(* IEC 61131-3 sources: com.logicals.lc3.webinar/logicals_Lib_Webinar/logicals_Webinar_Basic_Lib/logicals_Lib/src_FB_ST/Logic, 1 file *)

(* ---- logicals_Logic_ST.iecst ---- *)
NAMESPACE com.logicals.Basic.Logic

FUNCTION_BLOCK FB_lc_1oo3_ST

  VAR_INPUT
    vix_In1 : BOOL;
    vix_In2 : BOOL;
    vix_In3 : BOOL;
  END_VAR

  VAR_OUTPUT
   vox_Out : BOOL;
  END_VAR

  VAR
   lx_Var_AND1  : BOOL;
   lx_Var_AND2 : BOOL;
   lx_Var_AND3 : BOOL;
  END_VAR

  // Network 1:
  lx_Var_AND1 := AND(IN1 := vix_In1, IN2 := NOT vix_In2, IN3 := NOT vix_In3);
  lx_Var_AND2 := AND(IN1 := NOT vix_In1, IN2 := vix_In2, IN3 := NOT vix_In3);
  lx_Var_AND3 := AND(IN1 := NOT vix_In1, IN2 := NOT vix_In2, IN3 := vix_In3);
  vox_Out := OR(IN1 := lx_Var_AND1, IN2 := lx_Var_AND2, IN3 := lx_Var_AND3);

END_FUNCTION_BLOCK

FUNCTION_BLOCK FB_lc_1oo4_ST
	VAR_INPUT
		vix_In1 : BOOL;
		vix_In2 : BOOL;
		vix_In3 : BOOL;
		vix_In4 : BOOL;
	END_VAR

	VAR_OUTPUT
		vox_Out1 : BOOL;
		vox_Out2 : BOOL;
		vox_Out3 : BOOL;
		vox_Out4 : BOOL;

        vox_Err  : BOOL;
	END_VAR

    vox_Out1 := vix_In1 = TRUE  AND vix_In2 = FALSE AND vix_In3 = FALSE AND vix_In4 = FALSE;
    vox_Out2 := vix_In1 = FALSE AND vix_In2 = TRUE  AND vix_In3 = FALSE AND vix_In4 = FALSE;
    vox_Out3 := vix_In1 = FALSE AND vix_In2 = FALSE AND vix_In3 = TRUE  AND vix_In4 = FALSE;
    vox_Out4 := vix_In1 = FALSE AND vix_In2 = FALSE AND vix_In3 = FALSE AND vix_In4 = TRUE ;

    vox_Err :=  NOT(vox_Out1 = TRUE OR vox_Out2 = TRUE OR vox_Out3 = TRUE OR vox_Out4 = TRUE);

END_FUNCTION_BLOCK

FUNCTION_BLOCK FB_lc_1oo5_ST
	VAR_INPUT
		vix_In1 : BOOL;
		vix_In2 : BOOL;
		vix_In3 : BOOL;
		vix_In4 : BOOL;
		vix_In5 : BOOL;
	END_VAR

	VAR_OUTPUT
		vox_Out1 : BOOL;
		vox_Out2 : BOOL;
		vox_Out3 : BOOL;
		vox_Out4 : BOOL;
		vox_Out5 : BOOL;

        vox_Err  : BOOL;
	END_VAR

    vox_Out1 := vix_In1 = TRUE  AND vix_In2 = FALSE AND vix_In3 = FALSE AND vix_In4 = FALSE AND vix_In5 = FALSE;
    vox_Out2 := vix_In1 = FALSE AND vix_In2 = TRUE  AND vix_In3 = FALSE AND vix_In4 = FALSE AND vix_In5 = FALSE;
    vox_Out3 := vix_In1 = FALSE AND vix_In2 = FALSE AND vix_In3 = TRUE  AND vix_In4 = FALSE AND vix_In5 = FALSE;
    vox_Out4 := vix_In1 = FALSE AND vix_In2 = FALSE AND vix_In3 = FALSE AND vix_In4 = TRUE  AND vix_In5 = FALSE;
    vox_Out5 := vix_In1 = FALSE AND vix_In2 = FALSE AND vix_In3 = FALSE AND vix_In4 = FALSE AND vix_In5 = TRUE;

    vox_Err :=  NOT(vox_Out1 = TRUE OR vox_Out2 = TRUE OR vox_Out3 = TRUE OR vox_Out4 = TRUE OR vox_Out5 = TRUE );

END_FUNCTION_BLOCK

FUNCTION_BLOCK FB_lc_1oo6_ST
	VAR_INPUT
		vix_In1 : BOOL;
		vix_In2 : BOOL;
		vix_In3 : BOOL;
		vix_In4 : BOOL;
		vix_In5 : BOOL;
		vix_In6 : BOOL;
	END_VAR

	VAR_OUTPUT
		vox_Out1 : BOOL;
		vox_Out2 : BOOL;
		vox_Out3 : BOOL;
		vox_Out4 : BOOL;
		vox_Out5 : BOOL;
		vox_Out6 : BOOL;

        vox_Err  : BOOL;
	END_VAR

    vox_Out1 := vix_In1 = TRUE  AND vix_In2 = FALSE AND vix_In3 = FALSE AND vix_In4 = FALSE AND vix_In5 = FALSE AND vix_In6 = FALSE;
    vox_Out2 := vix_In1 = FALSE AND vix_In2 = TRUE  AND vix_In3 = FALSE AND vix_In4 = FALSE AND vix_In5 = FALSE AND vix_In6 = FALSE;
    vox_Out3 := vix_In1 = FALSE AND vix_In2 = FALSE AND vix_In3 = TRUE  AND vix_In4 = FALSE AND vix_In5 = FALSE AND vix_In6 = FALSE;
    vox_Out4 := vix_In1 = FALSE AND vix_In2 = FALSE AND vix_In3 = FALSE AND vix_In4 = TRUE  AND vix_In5 = FALSE AND vix_In6 = FALSE;
    vox_Out5 := vix_In1 = FALSE AND vix_In2 = FALSE AND vix_In3 = FALSE AND vix_In4 = FALSE AND vix_In5 = TRUE  AND vix_In6 = FALSE;
    vox_Out6 := vix_In1 = FALSE AND vix_In2 = FALSE AND vix_In3 = FALSE AND vix_In4 = FALSE AND vix_In5 = FALSE AND vix_In6 = TRUE;

    vox_Err :=  NOT(vox_Out1 = TRUE OR vox_Out2 = TRUE OR vox_Out3 = TRUE OR vox_Out4 = TRUE OR vox_Out5 = TRUE OR vox_Out6 = TRUE );

END_FUNCTION_BLOCK
 /*
  * Toogle per Eingang
  */
FUNCTION_BLOCK FB_lc_Toggle_ST
  /*
   * Toggle
   */
  VAR_INPUT
    /* Ein-Aus-Signal von SPS-Programm */
    vix_In : BOOL;
  END_VAR

  VAR_OUTPUT
    /* Ein-Aus-Signal als Status Toggle */
    vox_Out : BOOL;
  END_VAR
  /*
   * Baustein-Instanzen
   */
  VAR
    R_TRIG : R_TRIG;
  END_VAR

  VAR

  END_VAR

/*
 * SPS-Programmteil
 */
 R_TRIG(CLK:=vix_In);
 vox_Out:=XOR(R_TRIG.Q,vox_Out);

END_FUNCTION_BLOCK

 /*
  * ElTako
  * Toogle per Eingang
  */
FUNCTION_BLOCK FB_lc_ElTako_ST
  /*
   * Simulation eines ElTako-Relais
   */
  VAR_INPUT
    /* Ein-Aus-Signal von SPS-Programm */
    vix_In : BOOL;
  END_VAR

  VAR_OUTPUT
    /* Ein-Aus-Signal als Status ElTako */
    vox_Out : BOOL;
  END_VAR
  /*
   * Baustein-Instanzen
   */
  VAR
    R_TRIG : R_TRIG;
  END_VAR

  VAR

  END_VAR
/*
 * SPS-Programmteil
 */
 R_TRIG(CLK:=vix_In);
 vox_Out:=XOR(R_TRIG.Q,vox_Out);

END_FUNCTION_BLOCK

END_NAMESPACE
